Fanuc KAREL source: kx00008.KL

-- PROVISIONAL review KL for V770-1; original PC SHA256 7a213c5128099289852ba6156298965b6cb7123d54f231bb097ad9941aab5ecf
-- Incomplete behavior may be omitted. Consult companion uncertainty JSON. Do not deploy.
PROGRAM KX00008
%NOLOCKGROUP
VAR
  I : INTEGER
  J : INTEGER
  B : BOOLEAN
  F : FILE
  S : STRING[80]
-- UNRESOLVED_DECL P type=000102
BEGIN
  -- UNRESOLVED_PC offsets 5-7; opcodes 9C,3A
  -- UNRESOLVED_PC offsets 12-16; opcodes 7F
END KX00008
